{attribute 'reflection'} 
{attribute 'no_explicit_call' := 'do not call this POU directly'} 
FUNCTION_BLOCK FB_VAC_BLOW_VALVE IMPLEMENTS I_VAC_VALVE
VAR_INPUT
END_VAR
VAR_OUTPUT
END_VAR
VAR
	{attribute 'instance-path'} 
    {attribute 'noinit'} 
	strInstancePath: STRING;
	strFullObjectPath: STRING;
	stEvent: ST_EVENT;
	bAck: BOOL;
	itfOpMode:			I_OP_MODE;
	itfValveVac: I_BASE_VALVE;
	itfValveBlow: I_BASE_VALVE;
	itfSensorVacDetect: I_BINARY_SWITCH;

	
END_VAR

METHOD FB_init : BOOL
VAR_INPUT
	bInitRetains : BOOL; // if TRUE, the retain variables are initialized (warm start / cold start)
	bInCopyCode : BOOL;  // if TRUE, the instance afterwards gets moved into the copy code (online change)
	itfOpMode:			I_OP_MODE;
	itfValveVac: I_BASE_VALVE;
	itfValveBlow: I_BASE_VALVE;
	itfSensorVacDetect: I_BINARY_SWITCH;
END_VAR
THIS^.itfOpMode:= itfOpMode;
THIS^.itfValveVac:= itfValveVac;
THIS^.itfValveBlow:= itfValveBlow;
THIS^.itfSensorVacDetect:= itfSensorVacDetect;
END_METHOD

{warning 'Methodenimplementierung hinzufügen'}
METHOD M_AllOff
THIS^.itfValveVac.M_Close();
THIS^.itfValveBlow.M_Close();
END_METHOD

{warning 'Methodenimplementierung hinzufügen'}
METHOD M_Blow
THIS^.itfValveVac.M_Close();
THIS^.itfValveBlow.M_OPEN();
END_METHOD

{warning 'Methodenimplementierung hinzufügen'}
(*=== Method: M_Run  ============================================

 @brief: Here is the global code (Timer, Event, Flange,...)*)
METHOD M_Run
F_HandleInheritanceObjectInMRun(itfInheritanceObject:=THIS^.itfSensorVacDetect,itfThisObject:=THIS^);
F_HandleInheritanceObjectInMRun(itfInheritanceObject:=THIS^.itfValveVac,itfThisObject:=THIS^);
END_METHOD

{warning 'Methodenimplementierung hinzufügen'}
METHOD M_Vac
THIS^.itfValveVac.M_OPEN();
THIS^.itfValveBlow.M_Close();
END_METHOD


(*=== Property: P_Event  ============================================

 @param [set]: 	Set the Structure "ST_EVENT" from another Object
 @param [get]: 	Return the Structure "ST_EVENT", it contains the actual 
					event of the Object *)
PROPERTY P_Event : ST_EVENT
GET
P_Event:= stEvent;
END_GET
SET
END_SET
END_PROPERTY


(*=== Property: P_FullObjectPath  ============================================

 @param [set]: 	Set the Object Path (Clear String of Object)
 @param [get]: 	Return the Objectpath *)
PROPERTY P_FullObjectPath : STRING
GET
P_FullObjectPath:= THIS^.strFullObjectPath;
END_GET
SET
THIS^.strFullObjectPath:= P_FullObjectPath;
END_SET
END_PROPERTY


(*=== Property: P_Global_Ack  ============================================

 @param [set]: 	Set the Bit for Ack from another Object
 @param [get]: 	Return the state of Ack Bit*)
PROPERTY P_Global_Ack : BOOL
GET
P_Global_Ack:= THIS^.bAck;
END_GET
SET
THIS^.bAck:=P_Global_Ack;
END_SET
END_PROPERTY


(*=== Property: P_GlobalID  ============================================

 @param [set]: 	-
 @param [get]: 	Return the string of instance path*)
PROPERTY P_GlobalID : STRING
GET
P_GlobalID:= THIS^.strInstancePath;
END_GET
END_PROPERTY


PROPERTY P_STATE : E_PNEU_VAC_VALVE
GET
IF THIS^.itfValveVac.P_IS_OPEN THEN
	P_STATE:=E_PNEU_VAC_VALVE.Vac_ON_NotDetect;
END_IF

IF THIS^.itfValveVac.P_IS_CLOSE THEN
	P_STATE:=E_PNEU_VAC_VALVE.AllOff;
END_IF

IF THIS^.itfSensorVacDetect.P_Active THEN
	 P_STATE:=E_PNEU_VAC_VALVE.VacDetect;
 END_IF
 
 IF THIS^.itfValveBlow.P_IS_OPEN THEN
	 P_STATE:=E_PNEU_VAC_VALVE.Blowing;
 END_IF
END_GET
END_PROPERTY

END_FUNCTION_BLOCK

(* stored: Version 1.1.0.1, ProductVersion 3.1.4024.12
   POU FB_VAC_BLOW_VALVE: Id {458f9b90-019b-42cc-971a-ae9ac95c2d03}, SpecialFunc None
   Method FB_init: Id {1fd5d2b1-6119-4536-84f9-a2380392d3c1}
   Method M_AllOff: Id {d0932a76-ec6f-4d20-8e8b-67543967854b}
   Method M_Blow: Id {3e2280e5-035b-4a09-afb9-80da9a9c2559}
   Method M_Run: Id {b5565619-4816-4d27-bcab-82206a5ad576}
   Method M_Vac: Id {e0e7cf6a-03c5-4d17-9d8e-27cd1156242e}
   Property P_Event: Id {9b202751-d0ba-4fe1-9c94-59fa8212f0ba}
   Get Get: Id {30211a1f-16d1-4a96-a98a-00d2a2706495}
   Set Set: Id {267c0256-3ef0-4649-9adc-08addf285425}
   Property P_FullObjectPath: Id {ede7514b-60c3-44ca-bffd-edea0d8e65be}
   Get Get: Id {f82bab78-cdcb-4e17-aaa8-6a31d70be477}
   Set Set: Id {3845039a-ed5e-4c9d-90ab-17fdbd475ea8}
   Property P_Global_Ack: Id {d563e364-f937-4e4f-b2e1-e581109896c1}
   Get Get: Id {02a8c969-8729-4e77-a2e9-1499f51221e9}
   Set Set: Id {aa47cce3-a682-4551-9788-87efd1feffc8}
   Property P_GlobalID: Id {68a51acd-ad74-44de-a2e6-b2d1e1d55c09}
   Get Get: Id {f16a56b1-f028-4130-be1a-cde56eee44b5}
   Property P_STATE: Id {edeaf7f7-dbf6-4673-a144-79606a72f5df}
   Get Get: Id {8df11dae-8277-4d8d-8b37-9c32e8e0c41a} *)
